FUNCTION_BLOCK FB_ButtonBox
VAR_INPUT
	iInput1 : BOOL;
	iInput2 : BOOL;
	iInput3 : BOOL;
END_VAR
VAR_OUTPUT
	Q : BOOL;
	oLight1 : BOOL;	
END_VAR
VAR
	nState: eFeed;
	eTextWriteState : (OPEN_FILE, WRITE_TO_FILE, CLOSE_FILE, ERROR);
	Button1_trig: R_TRIG;
	Switch1_trig: R_TRIG;
	Switch2_trig: R_TRIG;
	tempCount1: INT;
	tempCount2: INT;
	tempCount3: INT;
	tempCount0: INT;
	
END_VAR

A_ButtonPressHandling();
A_Switch();


CASE nState OF
eFeed.Auto: 
		oLight1 := General.FastBlinkOn;
		
eFeed.Manual:
	IF Button1_trig.Q THEN
		nState := 2;
	END_IF
	
2:
		oLight1 := General.BlinkOn;
//	CLOSE_FILE:
		oLight1 := General.BlinkOn;		

END_CASE

ACTION A_ButtonPressHandling:
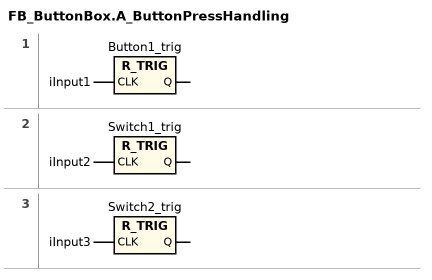
// NETWORK 1
Button1_trig(CLK := iInput1); // R_TRIG

// NETWORK 2
Switch1_trig(CLK := iInput2); // R_TRIG

// NETWORK 3
Switch2_trig(CLK := iInput3); // R_TRIG
END_ACTION

ACTION A_FeedButton:

END_ACTION

ACTION A_Switch:
IF General.ReadyForAction THEN
	IF Switch1_trig.Q THEN
	nState := 0;
	tempCount2 := tempCount2+1;
	END_IF
	IF Switch2_trig.Q THEN
	nState := 1;
	tempCount3 := tempCount3+1;
	END_IF
END_IF
END_ACTION

END_FUNCTION_BLOCK

(* stored: Version 1.1.0.1, ProductVersion 3.1.4024.10
   POU FB_ButtonBox: Id {718ab21c-a86f-42b1-ad84-7eea86241524}, SpecialFunc None
   Action A_ButtonPressHandling: Id {3b6590fa-f99a-41e5-8828-c964d473a0f6}
   Action A_FeedButton: Id {bbc46cfd-fa01-479f-b17d-06698f531804}
   Action A_Switch: Id {ab8781ab-cba4-40f4-9111-ef8f6611efbe} *)
